FUNCTION_BLOCK Tiefgarage
VAR_INPUT
END_VAR
VAR_OUTPUT
END_VAR
VAR
	Timer: TON;
END_VAR

//MAIN.Auto := 11;
//MAIN.Personen := 22;
DIO.DQ_1 := MAIN.B1;
DIO.DQ_2 := MAIN.B2;

Timer(IN:= NOT Timer.Q, PT:= T#10S );

END_FUNCTION_BLOCK

(* stored: Version 1.1.0.1, ProductVersion 3.1.4022.7
   POU Tiefgarage: Id {1b8e7ec7-cd2f-4faf-a8ae-b551aae7de3b}, SpecialFunc None *)
